// TIA Portal V16 export
// export: Created 2021-06-17T11:14:32.8951396Z, ExportSetting WithDefaults, DisplayName Totally Integrated Automation Portal, DisplayVersion V16 Update 4, DisplayName TIA Portal Version Control Interface, DisplayVersion V16 Update 2, DisplayName TIA Portal Openness, DisplayVersion V16 Update 4, DisplayName SINAMICS Startdrive Advanced, DisplayVersion V16 Update 5, DisplayName SINAMICS Startdrive G130, G150, S120, S150, SINAMICS MV, S210, DisplayVersion V16 Update 5, DisplayName SINAMICS Startdrive G110M, G120, G120C, G120D, G120P, G115D, DisplayVersion V16 Update 5, DisplayName STEP 7 Professional, DisplayVersion V16 Update 4, DisplayName SIMATIC Energy Suite, DisplayVersion V16 Update 4, DisplayName STEP 7 Safety, DisplayVersion V16, DisplayName WinCC Advanced / Unified PC, DisplayVersion V16 Update 4, DisplayName SIMATIC Visualization Architect, DisplayVersion V16 Update 1
VAR_GLOBAL   // PLC tag table "Default tag table"
   iL1 AT %IW2 : UInt;
   iL2 AT %IW4 : UInt;
   iL3 AT %IW6 : UInt;
   sTotal AT %IW8 : Int;
   qTotal AT %IW10 : Int;
   pTotal AT %IW12 : Int;
   reactEnTotal AT %ID18 : DInt;
   actEnTotal AT %ID14 : DInt;
   UserDataVar AT %IB0 : Byte;
   QualityInform AT %IB1 : Byte;
   pfTotal AT %IB23 : USInt;
   "Scaling current L1" AT %IB24 : USInt;
   "Scaling current L2" AT %IB25 : USInt;
   "Scaling current L3" AT %IB26 : USInt;
   "Scaling total active power L1L2L3" AT %IB27 : USInt;
   "Scaling total reactive power L1L2L3" AT %IB28 : USInt;
   "Scaling total apparent power L1L2L3" AT %IB29 : USInt;
   "Scaling total active energy L1L2L3" AT %IB30 : USInt;
   "Scaling total reactive energy L1L2L3" AT %IB31 : USInt;
END_VAR
